// Mitsubishi GX Works2 project: FB   PLC: Q02/Q02H

PROGRAM MAIN
VAR
  TEST_1 : TEST;
END_VAR
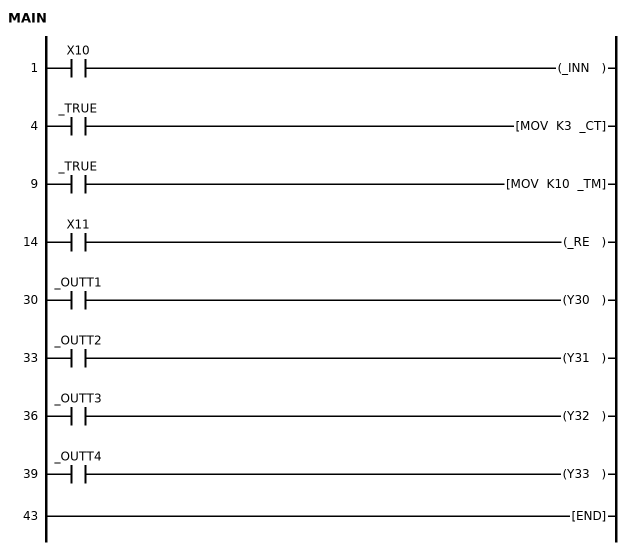
; FB BLK START TEST(TEST_1)
1     LD      X10
      OUT     _INN
4     LD      _TRUE
      MOV     K3 _CT
9     LD      _TRUE
      MOV     K10 _TM
14    LD      X11
      OUT     _RE
; FB START
; FB_NAME TEST
; INSTANCE_NAME TEST_1
; FB IN_B:INN
; FB OUT_OUTT1:B
; FB IN_W:CT
; FB OUT_OUTT2:B
; FB IN_W:TM
; FB OUT_OUTT3:B
; FB IN_B:RE
; FB OUT_OUTT4:B
; FB OUT_CTNUM:W
; FB END
30    LD      _OUTT1
      OUT     Y30
33    LD      _OUTT2
      OUT     Y31
36    LD      _OUTT3
      OUT     Y32
39    LD      _OUTT4
      OUT     Y33
; FB BLK END
43    END
END_PROGRAM

FUNCTION_BLOCK CTU
VAR_INPUT
  RE : BOOL;
  CU : BOOL;
  NUM : INT;
END_VAR
VAR_OUTPUT
  Q : BOOL;
END_VAR
VAR
  CNUM : INT;
END_VAR
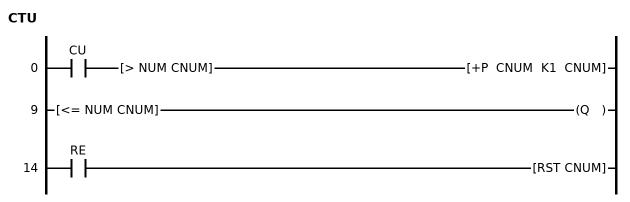
0     LD      CU
      AND>    NUM CNUM
      +P      CNUM K1 CNUM
9     LD<=    NUM CNUM
      OUT     Q
14    LD      RE
      RST     CNUM
END_FUNCTION_BLOCK

FUNCTION_BLOCK 인터록
VAR_INPUT
  INN1 : BOOL;
  INN2 : BOOL;
END_VAR
VAR_OUTPUT
  OUTT1 : BOOL;
  OUTT2 : BOOL;
END_VAR
VAR_INPUT
  INN3 : BOOL;
END_VAR
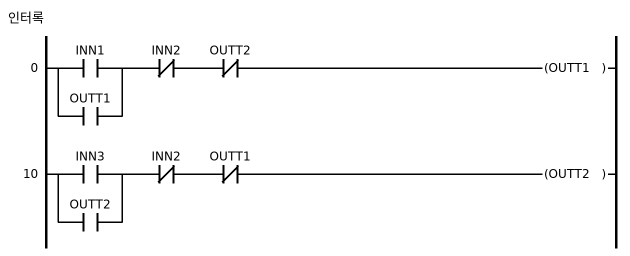
0     LD      INN1
      OR      OUTT1
      ANI     INN2
      ANI     OUTT2
      OUT     OUTT1
10    LD      INN3
      OR      OUTT2
      ANI     INN2
      ANI     OUTT1
      OUT     OUTT2
END_FUNCTION_BLOCK

FUNCTION_BLOCK 플리커
VAR_INPUT
  STT : BOOL;
  STP : BOOL;
END_VAR
VAR
  MM1 : BOOL;
END_VAR
VAR_INPUT
  PT1 : INT;
  PT2 : INT;
END_VAR
VAR_OUTPUT
  Q : BOOL;
  ET1 : INT;
  ET2 : INT;
END_VAR
VAR
  TT1 : TIMER;
  TT2 : TIMER;
END_VAR
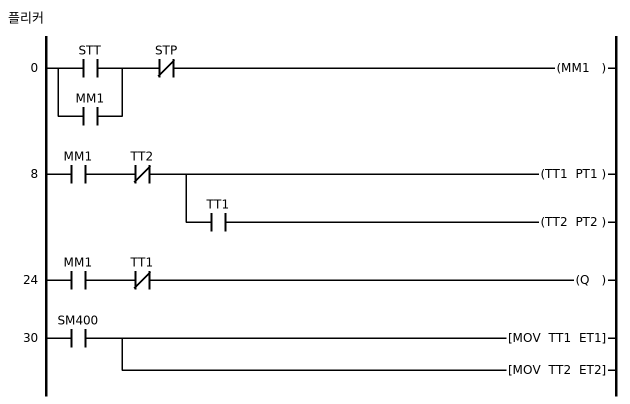
0     LD      STT
      OR      MM1
      ANI     STP
      OUT     MM1
8     LD      MM1
      ANI     TT2
      OUT     TT1 PT1
      AND     TT1
      OUT     TT2 PT2
24    LD      MM1
      ANI     TT1
      OUT     Q
30    LD      SM400
      MOV     TT1 ET1
      MOV     TT2 ET2
END_FUNCTION_BLOCK

FUNCTION_BLOCK 도장회로
VAR_INPUT
  ADV : BOOL;
  BACK : BOOL;
END_VAR
VAR_OUTPUT
  TEMP : BOOL;
END_VAR
VAR
  OUTT1 : BOOL;
END_VAR
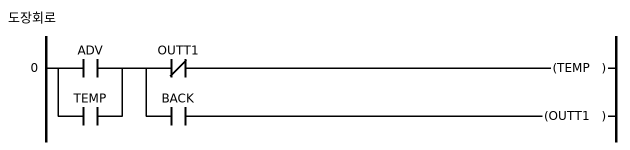
0     LD      ADV
      OR      TEMP
      MPS
      ANI     OUTT1
      OUT     TEMP
      MPP
      AND     BACK
      OUT     OUTT1
END_FUNCTION_BLOCK

FUNCTION_BLOCK CTD
VAR_INPUT
  INN : BOOL;
  RE : BOOL;
  CNUM : INT;
END_VAR
VAR_OUTPUT
  OUTT : BOOL;
  NOWNUM : INT;
END_VAR
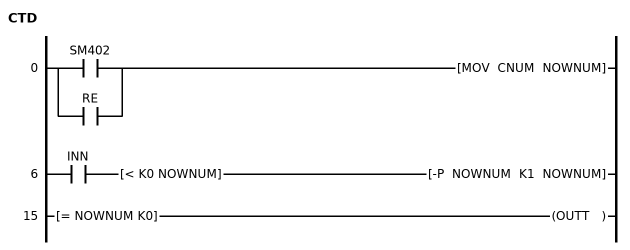
0     LD      SM402
      OR      RE
      MOV     CNUM NOWNUM
6     LD      INN
      AND<    K0 NOWNUM
      -P      NOWNUM K1 NOWNUM
15    LD=     NOWNUM K0
      OUT     OUTT
END_FUNCTION_BLOCK

FUNCTION_BLOCK TEST
VAR_INPUT
  INN : BOOL;
  CT : INT;
END_VAR
VAR_OUTPUT
  OUTT1 : BOOL;
  OUTT2 : BOOL;
  OUTT3 : BOOL;
  OUTT4 : BOOL;
END_VAR
VAR_INPUT
  TM : INT;
  RE : BOOL;
END_VAR
VAR_OUTPUT
  CTNUM : INT;
END_VAR
VAR
  TT1 : TIMER;
  TT2 : TIMER;
  TT3 : TIMER;
  TT4 : TIMER;
  CT1 : COUNTER;
  MM1 : BOOL;
END_VAR
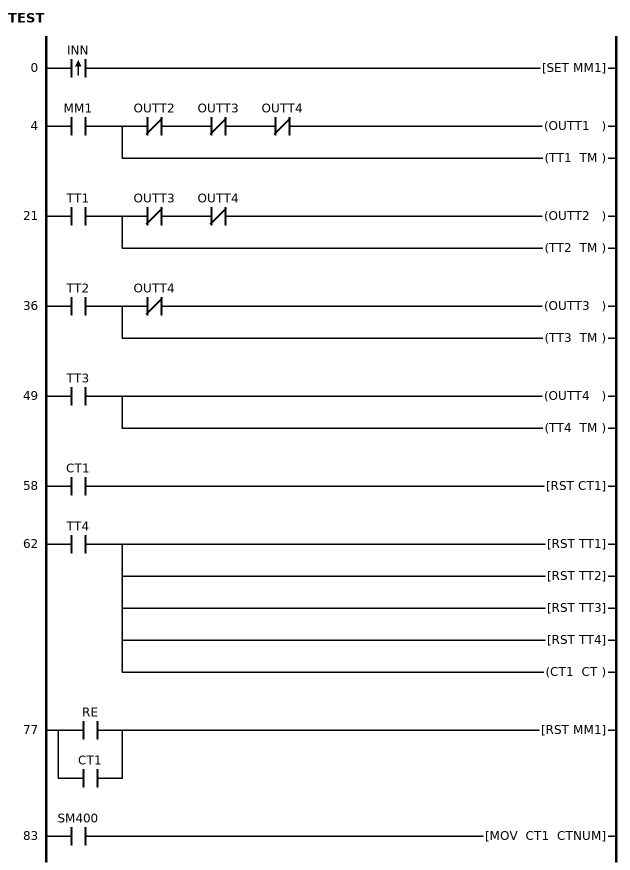
0     LDP     INN
      SET     MM1
4     LD      MM1
      MPS
      ANI     OUTT2
      ANI     OUTT3
      ANI     OUTT4
      OUT     OUTT1
      MPP
      OUT     TT1 TM
21    LD      TT1
      MPS
      ANI     OUTT3
      ANI     OUTT4
      OUT     OUTT2
      MPP
      OUT     TT2 TM
36    LD      TT2
      MPS
      ANI     OUTT4
      OUT     OUTT3
      MPP
      OUT     TT3 TM
49    LD      TT3
      OUT     OUTT4
      OUT     TT4 TM
58    LD      CT1
      RST     CT1
62    LD      TT4
      RST     TT1
      RST     TT2
      RST     TT3
      RST     TT4
      OUT     CT1 CT
77    LD      RE
      OR      CT1
      RST     MM1
83    LD      SM400
      MOV     CT1 CTNUM
END_FUNCTION_BLOCK
